// TIA Portal V18 export
VAR_GLOBAL   // PLC tag table "Sirena"
   sir_1 AT %Q32.0 : Bool;
   sir_2 AT %Q32.1 : Bool;
   sir_3 AT %Q32.2 : Bool;
   sir_4 AT %Q32.3 : Bool;
   sir_5 AT %Q33.0 : Bool;
   sir_6 AT %Q33.1 : Bool;
   sir_start AT %Q33.2 : Bool;
END_VAR
